// TIA Portal V20 export
DATA_BLOCK "STATION"   // DB130
{ S7_Optimized_Access := 'FALSE' }
VERSION : 0.1
// stored: AutoNumber false, DBAccessibleFromOPCUA true, DBAccessibleFromWebserver false, IsOnlyStoredInLoadMemory false, IsWriteProtectedInAS false
   VAR RETAIN
      Count : UInt;
      Station { S7_SetPoint := 'True'} : Array["STATION_MIN".."STATION_MAX"] of "LGR_STATION";
      InterlockByGRM { S7_SetPoint := 'True'} : Array["STATION_MIN".."STATION_MAX"] of "LGR_Interface_CV_PO";
      PreData : Struct
         Tracking : Array["STATION_MIN".."STATION_MAX"] of "LGR_Station_TrackingData";
         Error { S7_SetPoint := 'True'} : Array["STATION_MIN".."STATION_MAX"] of "LGR_Station_TrackingData";
         Last { S7_SetPoint := 'True'} : Array["STATION_MIN".."STATION_MAX"] of "LGR_Station_TrackingData";
      END_STRUCT;
   END_VAR
BEGIN
END_DATA_BLOCK
